FUNCTION_BLOCK RollingFille
VAR
	state : RollingFileState;
	file_open : Tc2_System.FB_FileOpen;
	file_close : Tc2_System.FB_FileClose;
	file_write : Tc2_System.FB_FileWrite;
	file_handle : UINT;

	file_name : Tc2_System.T_MaxString; // File name including its path

	lockFileWriteToForceRisingEdge : BOOL; // filePuts can only be executed every other cycle
									 // since it needs a rising edge to execute.
	
END_VAR

PROPERTY PUBLIC IsClosed : BOOL
GET // PUBLIC
IsClosed := state = RollingFileState.Closed;
END_GET
END_PROPERTY

PROPERTY PUBLIC IsOpen : BOOL
GET // PUBLIC
IsOpen := state = RollingFileState.Open;
END_GET
END_PROPERTY

METHOD PRIVATE OnOpenState
VAR_INPUT
END_VAR
END_METHOD

METHOD PUBLIC Open : BOOL
VAR_INPUT
END_VAR
file_open(
	sNetId := '',
	sPathName := file_name,
	nMode := FOPEN_MODEAPPEND OR FOPEN_MODETEXT, 
	ePath := PATH_GENERIC,
	tTimeout := timeout,
	hFile => file_handle
);
END_METHOD

END_FUNCTION_BLOCK

(* stored: Version 1.1.0.1
   POU RollingFille: Id {fb0c942f-e725-4213-95a9-4aefd0bdfe94}, SpecialFunc None
   Property IsClosed: Id {475f4d6d-f6b8-4cac-9b30-844c2d7f8656}
   Get Get: Id {25e5d962-2214-4a21-922c-a892ffbbde5d}
   Property IsOpen: Id {0a125925-6eda-409f-bf72-b73719a2cea1}
   Get Get: Id {352c700f-c2e1-4ab7-b83c-7ae9bceef20e}
   Method OnOpenState: Id {7934a996-6792-4dc6-9b85-64947639d6fb}
   Method Open: Id {1513242a-6101-442a-a550-ffa27a32becc} *)
